// TwinCAT 3 PLC project OEf_3
// ProgramVersion: 3.1.4024.0
// libraries:
//   Tc2_Standard, * (Beckhoff Automation GmbH)
//   Tc2_System, * (Beckhoff Automation GmbH)
//   Tc3_Module, * (Beckhoff Automation GmbH)
// project tree:
//   / PlcTask.TcTTO
//   POUs/ MAIN.TcPOU
// (motion and I/O tree: see PLC project oef_1)
// real-time tasks:
//   TASK PlcTask: cycle T#10ms, priority 20, ADS port 350
//   TASK PlcTask1: cycle T#10ms, priority 21, ADS port 351
//   TASK PlcTask2: cycle T#10ms, priority 22, ADS port 352
// variable links:
//   OEf_3/OEf_3 Instance <-> Device 1 (EtherCAT)/Term 1 (EK1200)/Term 2 (EL1008)
//     PlcTask Inputs/MAIN.SW{2..5} <-> Channel {1..4}/Input  (4 links)
//   OEf_3/OEf_3 Instance <-> Device 1 (EtherCAT)/Term 1 (EK1200)/Term 3 (EL2008)
//     PlcTask Outputs/MAIN.Alarm <-> Channel 5/Output
//     PlcTask Outputs/MAIN.Orange <-> Channel 1/Output
//     PlcTask Outputs/MAIN.Rood <-> Channel 2/Output

CONFIGURATION OEf_3
    RESOURCE PLC ON TwinCAT3
        TASK PlcTask(INTERVAL := T#10ms, PRIORITY := 22);
        PROGRAM MAIN WITH PlcTask : MAIN;
    END_RESOURCE
END_CONFIGURATION

// ---- POUs/MAIN.TcPOU
PROGRAM MAIN
VAR
	Rood AT %Q*: BOOL := FALSE;
	Orange AT %Q*: BOOL := false;
	Alarm AT %Q*: BOOL := FALSE;
	Headswitch AT %I*: BOOL := true;
	SW3 AT %I*: BOOL := false;
	SW4 AT %I*: BOOL := false;
	SW5 AT %I*: BOOL := false;
	SW2 AT %I*: BOOL := false;
END_VAR

Orange := Headswitch AND (SW3 OR SW4 OR SW5)AND (NOT SW2);
Rood := Headswitch AND ((SW3 AND SW4) OR (SW3 AND SW5) OR (SW4 AND SW5))AND (NOT SW2);
Alarm := Headswitch AND SW3 AND SW4 AND SW5 AND (NOT SW2);

END_PROGRAM
